FUNCTION_BLOCK RejectArmController
  (* Standard: 61499-2 *)
  (* Version 0.1, 2016-00-28, hpea485, UOA *)
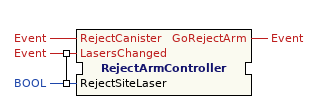
  EVENT_INPUT
    RejectCanister;
    LasersChanged WITH RejectSiteLaser;
  END_EVENT
  EVENT_OUTPUT
    GoRejectArm;
  END_EVENT
  VAR_INPUT
    RejectSiteLaser : BOOL;
  END_VAR
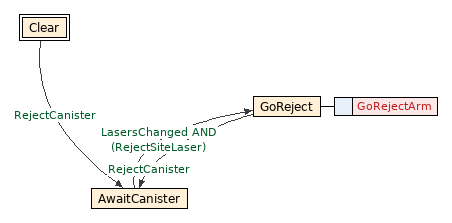
  EC_STATES
    Clear;
    AwaitCanister;
    GoReject : -> GoRejectArm;
  END_STATES
  EC_TRANSITIONS
    Clear TO AwaitCanister := RejectCanister;
    AwaitCanister TO GoReject := LasersChanged AND (RejectSiteLaser);
    GoReject TO AwaitCanister := RejectCanister;
  END_TRANSITIONS
END_FUNCTION_BLOCK
